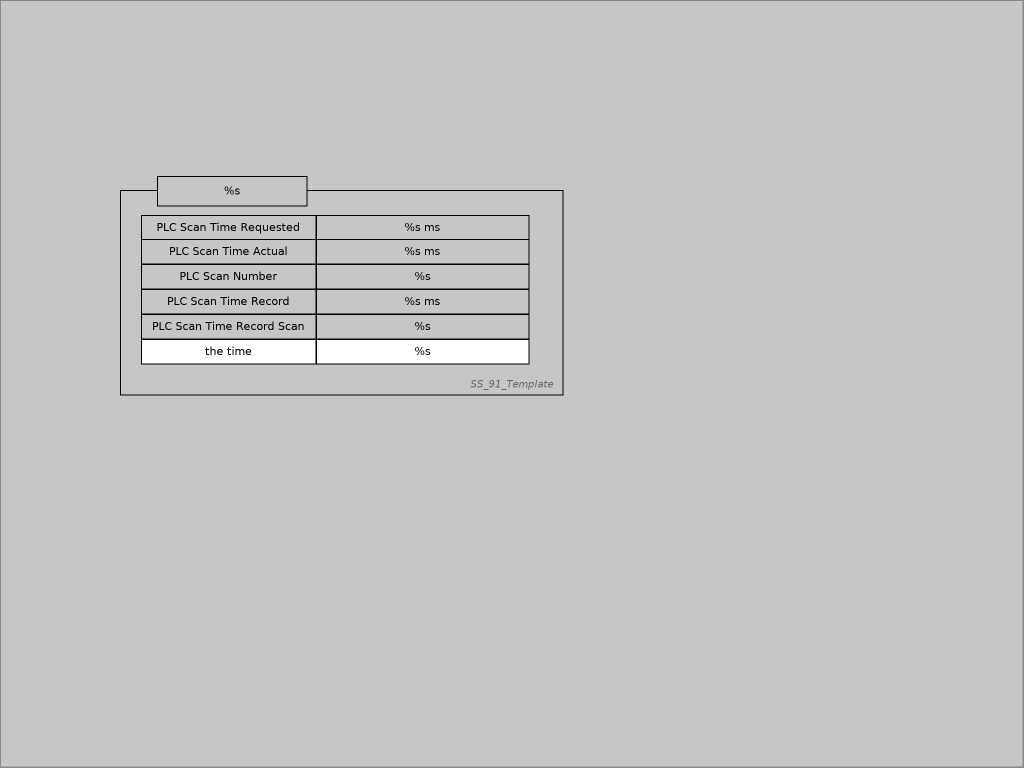
VISUALIZATION SS_11_HMISystem  // 1024x768
    Frame (0,0 1024x768)
        shows SS_91_Template(header := HMIData.hmiHeader)
    Rectangle (316,215 213x25), "%s ms", text variable: System.ScanTimeReq, text list: ''
    Rectangle (141,215 175x25), "PLC Scan Time Requested"
    Rectangle (141,239 175x25), "PLC Scan Time Actual"
    Rectangle (316,239 213x25), "%s ms", text variable: System.ScanTimeAct, text list: ''
    Rectangle (141,264 175x25), "PLC Scan Number"
    Rectangle (316,264 213x25), "%s", text variable: System.myPlcInfoTask1.CycleCount, text list: ''
    Rectangle (120,190 443x205)
    Rectangle (157,176 150x30), "%s", text variable: System.myPlcInfoTask1.TaskName
    Rectangle (141,289 175x25), "PLC Scan Time Record"
    Rectangle (316,289 213x25), "%s ms", text variable: System.ScanTimeRecord, text list: ''
    Rectangle (141,314 175x25), "PLC Scan Time Record Scan"
    Rectangle (316,314 213x25), "%s", text variable: System.ScanTimeRecordScan, text list: ''
    Rectangle (316,339 213x25), "%s", text variable: System.timeDT
    Rectangle (141,339 175x25), "the time"
END_VISUALIZATION

(* stored: Version 1.1.0.1, ProductVersion 3.1.4024.12
   Visu SS_11_HMISystem: Id {785d049b-80ed-4444-aba2-927731f3e4a5} *)
